PROGRAM MAIN
VAR
END_VAR

//TcUnit.RUN();

END_PROGRAM

(* stored: Version 1.1.0.1, ProductVersion 3.1.4024.12
   POU MAIN: Id {7e4abf7d-f388-0143-26ed-b64153253fe1}, SpecialFunc None *)
